{attribute 'GeneratedUsingTerminal: EK1200-1388-0000'}
{attribute addProperty BoxType "EK1200-1388-0000"}
{attribute addProperty Id "Term_2_EL6002EL6002_CD897635118Term_3_EL1809EL1809_32157CFD20Term_4_EL2809EL2809_2B6483BD19Term_5_EL4004EL4004_E203F87511Term_6_EL2809EL2809_2B6483BD19Term_7_EL6001EL6001_0DE01E7E61"}
{attribute addProperty CRC "4137248816"}
{attribute addProperty Size "248"}
TYPE Term_1_EK1200_F6996830 :
STRUCT
	{attribute addProperty Name "Term_2_EL6002"}
	{attribute addProperty PreviousPort "Term 1 (EK1200) : B"}
	Term_2_EL6002 : EL6002_CD897635;
	{attribute addProperty Name "Term_3_EL1809"}
	{attribute addProperty PreviousPort "Term 2 (EL6002) : B"}
	Term_3_EL1809 : EL1809_32157CFD;
	{attribute addProperty Name "Term_4_EL2809"}
	{attribute addProperty PreviousPort "Term 3 (EL1809) : B"}
	Term_4_EL2809 : EL2809_2B6483BD;
	{attribute addProperty Name "Term_5_EL4004"}
	{attribute addProperty PreviousPort "Term 4 (EL2809) : B"}
	Term_5_EL4004 : EL4004_E203F875;
	{attribute addProperty Name "Term_6_EL2809"}
	{attribute addProperty PreviousPort "Term 5 (EL4004) : B"}
	Term_6_EL2809 : EL2809_2B6483BD;
	{attribute addProperty Name "Term_7_EL6001"}
	{attribute addProperty PreviousPort "Term 6 (EL2809) : B"}
	Term_7_EL6001 : EL6001_0DE01E7E;
END_STRUCT
END_TYPE

(* stored: Version 1.2.0.0, ProductVersion 3.1.4024.9
   DUT Term_1_EK1200_F6996830: Id {743e5612-9d0e-0a1a-2e35-fbb3788af67b} *)
